{attribute 'no_explicit_call' := 'do not call this POU directly, call execute'} 
FUNCTION_BLOCK _TemplateFB
VAR
END_VAR

// NO CODE HERE, USE execute

METHOD execute
END_METHOD

END_FUNCTION_BLOCK

(* stored: Version 1.1.0.1
   POU _TemplateFB: Id {5b3ac5df-9d93-4b84-8bff-2d4073da45ad}, SpecialFunc None
   Method execute: Id {f125a433-0a62-494c-b1c6-308ef7e187e2} *)
